// TIA Portal V20 export
DATA_BLOCK "T5 EXCENTRIC HMI"   // DB1218
{ S7_Optimized_Access := 'TRUE' }
AUTHOR : SAS
// stored: AutoNumber false, IsRetainMemResEnabled true, MemoryReserve 100, RetainMemoryReserve 100
   VAR
      Conditions : Struct
         CG : "Pop_Up_Aux";   // General conditions
         CA : "Pop_Up_Aux";   // Start Auto mode conditions
         SC_Initial : "Pop_Up_Aux";   // Start cycle conditions
         SC_Vertical : "Pop_Up_Aux";   // Start cycle conditions
         MOV_FW : "Pop_Up_Aux";   // Movement interlocks Forward
         MOV_BW : "Pop_Up_Aux";   // Movement interlocks Backward
      END_STRUCT;
      HMI : Struct
         PB : Struct
            s0 : Bool;
            s1 : Bool;
            s2 : Bool;
            s3 : Bool;
            s4 : Bool;
            Pause : Bool;   // Pause
            s6 : Bool;
            s7 : Bool;
            s8 : Bool;
            s9 : Bool;
            s10 : Bool;
            s11 : Bool;
            s12 : Bool;
            s13 : Bool;
            s14 : Bool;
            s15 : Bool;
         END_STRUCT;
         ST : Struct
            s0 : Bool;
            s1 : Bool;
            s2 : Bool;
            s3 : Bool;
            s4 : Bool;
            Pause : Bool;   // Pause
            s6 : Bool;
            s7 : Bool;
            s8 : Bool;
            s9 : Bool;
            "ST Machine" : Int;   // Device label status (0=EME, 1=Safe, 2=Fault, 3=Run, 4=Stopped)
            "ST Sequencer step" : Int;   // Sequencer step
         END_STRUCT;
      END_STRUCT;
   END_VAR
BEGIN
   // Conditions.CG.Conditions.n1 : Tensiune Alimentare OK
   // Conditions.CG.Conditions.n2 : Electric protectie OK
   // Conditions.CG.Conditions.n3 : Inverter OK
   // Conditions.CA.Conditions.n1 : Conditiie Generale
   // Conditions.CA.Conditions.n2 : Excentric initial/vertical
   // Conditions.SC_Initial.Conditions.n1 : Initial Conditions
   // Conditions.SC_Initial.Conditions.n2 : Piece Presence
   // Conditions.SC_Initial.Conditions.n3 : Tracking OK
   // Conditions.SC_Initial.Conditions.n4 : Condition of movement
   // Conditions.SC_Initial.Conditions.n5 : T5 Role-1 Stopped
   // Conditions.SC_Initial.Conditions.n6 : T5 Lant Stopped and Home
   // Conditions.SC_Initial.Conditions.n7 : T5 Lant Free
   // Conditions.SC_Initial.Conditions.n8 : T5 Lant a facut un pas
   // Conditions.SC_Vertical.Conditions.n1 : Vertical Conditions
   // Conditions.SC_Vertical.Conditions.n2 : Condition of movement vertical
   // Conditions.SC_Vertical.Conditions.n3 : Tracking OK
   // Conditions.SC_Vertical.Conditions.n4 : T5 Lant Stopped and Home
   // Conditions.SC_Vertical.Conditions.n5 : T5 Lant Free
   // Conditions.SC_Vertical.Conditions.n6 : T5 Lant a facut un pas
   // Conditions.MOV_FW.Conditions.n1 : Permanent Conditions
   // Conditions.MOV_BW.Conditions.n1 : Permanent Conditions
END_DATA_BLOCK
